{attribute 'linkalways'} 
{attribute 'no_explicit_call' := 'This FB is a CLASS and must be accessed using methods or properties'}
{attribute 'enable_dynamic_creation'}
FUNCTION_BLOCK _TOD EXTENDS DatatypeBase
VAR
	localData : TOD;
	activeData : REFERENCE TO TOD REF= localData;
END_VAR

PROPERTY PUBLIC Address : PVOID
GET
Address := ADR(activeData);
END_GET
END_PROPERTY

METHOD PUBLIC ClearReference
VAR_INPUT
END_VAR
activeData REF= localData;
END_METHOD

METHOD PUBLIC Clone : I_Datatype
VAR
    pClone : POINTER TO _TOD;
END_VAR
pClone := __NEW(_TOD(InitialValue := Value));
Clone := pClone^;
END_METHOD

METHOD FB_init : BOOL
VAR_INPUT
	bInitRetains : BOOL; // if TRUE, the retain variables are initialized (warm start / cold start)
	bInCopyCode : BOOL;  // if TRUE, the instance afterwards gets moved WORDo the copy code (online change)
	InitialValue : TOD;
END_VAR
localData := InitialValue;
END_METHOD

METHOD PUBLIC MakeReferenceTo
VAR_INPUT
	ReferenceTarget : REFERENCE TO TOD;
END_VAR
activeData REF= ReferenceTarget;
END_METHOD

METHOD PUBLIC SerializeWith
VAR_INPUT
	Serializer : I_Serializer;
END_VAR
Serializer.AddTod(activeData);
END_METHOD

PROPERTY PUBLIC Size : UDINT
GET
Size := SIZEOF(activeData);
END_GET
END_PROPERTY

METHOD TryDeserializeFrom : BOOL
VAR_INPUT
	Deserializer : I_Deserializer;
	Feedback : I_DeserializerFeedback;
END_VAR
TryDeserializeFrom := Deserializer.TryGetTod(activeData, Feedback);
END_METHOD

METHOD TryMakeReferenceTo : BOOL
VAR_INPUT
	Target : I_Datatype;
END_VAR
VAR
	pTargetData : POINTER TO TOD;
END_VAR
IF NOT (Target.TypeName = TypeName) THEN
	RETURN;
END_IF

pTargetData := Target.Address;
activeData REF= pTargetData^;
TryMakeReferenceTo := TRUE;
END_METHOD

PROPERTY PUBLIC TypeName : T_MAXSTRING
GET
TypeName := 'TOD';
END_GET
END_PROPERTY

PROPERTY PUBLIC Value : REFERENCE TO TOD
GET
Value REF= activeData;
END_GET
END_PROPERTY

END_FUNCTION_BLOCK

(* stored: Version 1.1.0.1, ProductVersion 3.1.4024.12
   POU _TOD: Id {14577ba8-48ab-4051-ba80-c9e6931d7791}, SpecialFunc None
   Folder Constructor: Id {404083ff-f402-4987-8bb1-d846d67104aa}
   Property Address: Id {b1e4b8df-ce60-440d-a9ce-76da1e98bde1}
   Get Get: Id {761b471f-ccab-4b56-b768-93e430566d5a}
   Method ClearReference: Id {88237940-e3b3-45c2-9ad0-d645ca9cd45e}
   Method Clone: Id {92107c97-2d1e-480a-8969-907840f0b0db}
   Method FB_init: Id {5dec047b-587e-41bd-b5dd-c30f372d594b}
   Method MakeReferenceTo: Id {b90e1b8a-dad8-4343-addd-9efd3dcf7277}
   Method SerializeWith: Id {2b3fb066-e1b8-4763-beb0-aa0bfd2bf67c}
   Property Size: Id {809c2bcd-2901-4f24-8526-292992113fc4}
   Get Get: Id {66a79684-6ae9-42e3-9dca-504a0a63e004}
   Method TryDeserializeFrom: Id {065e51b7-1628-4c24-8c8d-8b12d9eb6424}
   Method TryMakeReferenceTo: Id {a03512e4-d20f-46b0-b391-f34d80a8b191}
   Property TypeName: Id {e9c7e272-6a59-4092-844e-bf847ed35fd5}
   Get Get: Id {79b12e39-c031-4bfe-8d6a-620ac0acff64}
   Property Value: Id {380c4051-aba4-4700-bb4d-797516b9c5ad}
   Get Get: Id {e4ae82f1-b88f-49ec-ae70-5b419277bbae} *)
